TYPE sAI_SCALE :
STRUCT
	rawLo: DINT := 0;
	rawHi: DINT := 32767;
	pvLo: LREAL := 0.0;
	pvHi: LREAL := 100.0;
	eu: STRING[20] := '%';
END_STRUCT
END_TYPE

(* stored: Version 1.1.0.1, ProductVersion 3.1.0.36
   DUT sAI_SCALE: Id {13a79b9c-b610-4891-a145-99a94036c64b} *)
